{attribute 'GeneratedUsingTerminal: EJ7211-0011-0026'}
{attribute addProperty BoxType "EJ7211-0011-0026"}
{attribute addProperty Id "ControlwordAT %Q*UINT2"}
{attribute addProperty CRC "4092675873"}
{attribute addProperty Size "2"}
TYPE DS402_Controlword_F3F14721 :
STRUCT
	{attribute addProperty Name "Controlword"}
	Controlword AT %Q* : UINT;
END_STRUCT
END_TYPE

(* stored: Version 1.2.0.0, ProductVersion 3.1.4024.9
   DUT DS402_Controlword_F3F14721: Id {75da181d-df3f-427b-9045-f5db1f207386} *)
